RESOURCE_TYPE _pizza
  (* Standard: 61499-2 *)
  (* Version 0.1, 2017-00-12, hpea485, UOA *)
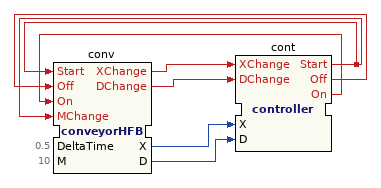
  FBS
    conv : conveyorHFB(DeltaTime := 0.5, M := 10);
    cont : controller;
  END_FBS
  EVENT_CONNECTIONS
    conv.XChange TO cont.XChange;
    conv.DChange TO cont.DChange;
    cont.Start TO conv.Start;
    cont.Start TO conv.MChange;
    cont.Off TO conv.Off;
    cont.On TO conv.On;
  END_CONNECTIONS
  DATA_CONNECTIONS
    conv.X TO cont.X;
    conv.D TO cont.D;
  END_CONNECTIONS
END_RESOURCE_TYPE
